// TIA Portal V19 export
TYPE "Prod_Halted_Str"
// stored: Access Published
   STRUCT
      Code : Int;   // Codice stato interruzione vedere tabella "Prod_Halted_Status_CONST"
      Detail : String;   // Dettaglio causa interruzione
   END_STRUCT;
END_TYPE
